// TwinCAT 3 PLC project PLC1
// ProgramVersion: 3.1.4023.0
// libraries:
//   Tc2_Standard, * (Beckhoff Automation GmbH)
//   Tc2_System, * (Beckhoff Automation GmbH)
//   Tc3_Module, * (Beckhoff Automation GmbH)
// project tree:
//   / Class Diagram.TcCD (not stored), Param.TcGVL, PlcTask.TcTTO
//   FBs/ FB_Colleague.TcPOU, FB_Mediator.TcPOU
//   ITFs/ I_Colleague.TcIO, I_Mediator.TcIO
//   POUs/ MAIN.TcPOU

CONFIGURATION PLC1
    RESOURCE PLC ON TwinCAT3
        TASK PlcTask(INTERVAL := T#10ms, PRIORITY := 20);
        PROGRAM MAIN WITH PlcTask : MAIN;
    END_RESOURCE
END_CONFIGURATION

// ---- Param.TcGVL
{attribute 'qualified_only'}
VAR_GLOBAL CONSTANT
	MAX_COLLEAGUES : INT := 6;
END_VAR

// ---- ITFs/I_Colleague.TcIO
INTERFACE I_Colleague

METHOD operation : BOOL
VAR_INPUT
	// Event string
	event : STRING;
END_VAR
END_METHOD

END_INTERFACE

// ---- ITFs/I_Mediator.TcIO
INTERFACE I_Mediator

METHOD notify : BOOL
VAR_INPUT
	// Colleague sending the notification
	sender : I_Colleague;
	// Some event the collegue is attempting
	event	  : STRING;
END_VAR
END_METHOD

END_INTERFACE

// ---- POUs/MAIN.TcPOU
PROGRAM MAIN
VAR
	fbChatWindow : FB_Mediator;
	fbUsers	     : ARRAY[1..Param.MAX_COLLEAGUES] OF FB_Colleague;
	
	ChatWindow	 : I_Mediator;
	Users		 : ARRAY[1..Param.MAX_COLLEAGUES] OF I_Colleague;
	
	// Task and Demo Control
	bStartDemo	: BOOL := TRUE;
	i: INT;
END_VAR

// Initialize Interface to Mediator
ChatWindow := fbChatWindow;
// Assign Users 
fbChatWindow(iColleague := Users);
FOR i := 1 TO Param.MAX_COLLEAGUES DO
	// Initialize Interface to Colleagues
	Users[i] := fbUsers[i];
	// Assign Mediator to Colleagues
	fbUsers[i](iMediator := ChatWindow);
END_FOR


IF bStartDemo THEN
	bStartDemo := FALSE;
	Users[1].operation('Hi! How is everyone?');
	Users[2].operation('Good good..');
	Users[4].operation('Doing fine');
	Users[5].operation('Yup! All is well');
	Users[3].operation('I need a beer right about now');
	Users[6].operation('Had a long day?');	
	Users[3].operation('Yuuup, very long...');
END_IF

END_PROGRAM

// ---- FBs/FB_Mediator.TcPOU
FUNCTION_BLOCK FB_Mediator IMPLEMENTS I_Mediator
VAR_INPUT
	iColleague : ARRAY [1..Param.MAX_COLLEAGUES] OF I_Colleague; // Colleague Interface Array
END_VAR

METHOD notify : BOOL
VAR_INPUT
	(* Colleague sending the notification*)
	sender	: I_Colleague;
	(* Some event the collegue is attempting*)
	event	: STRING;
END_VAR

VAR
	i: INT;
END_VAR
FOR i := 1 TO Param.MAX_COLLEAGUES DO
		IF iColleague[i] <> 0 AND iColleague[i] = sender THEN
			ADSLOGSTR(msgCtrlMask := ADSLOG_MSGTYPE_MSGBOX, msgFmtStr := CONCAT(CONCAT('User ', TO_STRING(i)), ' said: %s'), strArg := event);
		END_IF
END_FOR
END_METHOD

END_FUNCTION_BLOCK

// ---- FBs/FB_Colleague.TcPOU
FUNCTION_BLOCK FB_Colleague IMPLEMENTS I_Colleague
VAR_INPUT
	iMediator : REFERENCE TO I_Mediator; // Mediator Interface
END_VAR

METHOD operation : BOOL
VAR_INPUT
	event : STRING;
END_VAR
IF __ISVALIDREF(iMediator) THEN
	iMediator.notify(THIS^,event);
END_IF
END_METHOD

END_FUNCTION_BLOCK
